FUNCTION_BLOCK FB_MMSensor_full
VAR_INPUT
		lettura			:INT;
		distanzaAVuoto	:INT; 
		valSoglia		:INT;
		filterTime		:INT;		//seconds
END_VAR
VAR_OUTPUT
		full			:BOOL;
END_VAR
VAR
		_tmr			:TON;
		_over			:BOOL;
END_VAR



IF lettura < valSoglia THEN
	_over := TRUE;
ELSE
	_over:=FALSE;
	full:=FALSE;
END_IF

_tmr(IN:=_over, PT:=INT_TO_TIME(filterTime*1000));
IF _tmr.Q THEN
	_over:=FALSE;
	full:=TRUE;
END_IF

END_FUNCTION_BLOCK

(* stored: Version 1.1.0.1, ProductVersion 3.1.4022.12
   POU FB_MMSensor_full: Id {3e95e641-4c97-4606-bdf8-2bce40853b16}, SpecialFunc None *)
